FUNCTION F_CheckAxisLEQ : BOOL
VAR_INPUT
    stMotionStage: ST_MotionStage;
    fQueryValue: LREAL;
END_VAR
VAR
END_VAR


F_CheckAxisLEQ := F_CheckAxis(stMotionStage, 1, fQueryValue);

END_FUNCTION

(* stored: Version 1.1.0.1, ProductVersion 3.1.4022.18
   POU F_CheckAxisLEQ: Id {7e8f22ef-8fcc-4623-84e5-bac5a0ddc160}, SpecialFunc None *)
